INTERFACE I_ErrorVisitor

METHOD VisitError
VAR_INPUT
	VisitingError : I_Error;
END_VAR
END_METHOD

END_INTERFACE

(* stored: Version 1.1.0.1, ProductVersion 3.1.4024.12
   Itf I_ErrorVisitor: Id {129ca6d0-5a1c-05dc-0ec9-5aa9c0681d3c}
   Method VisitError: Id {e2c761d6-f0af-08c5-1c63-f5fdb44c6866} *)
